(* IEC 61131-3 sources: AXOpen/src/components.kuka.robotics/ctrl/src/AxoKukaRobotics_Datatypes_v_5_x_x, 9 files *)

(* ---- AxoKukaRobotics_Component_Status.st ---- *)
NAMESPACE AXOpen.Components.Kuka.Robotics.v_5_x_x
    {S7.extern=ReadWrite}
    {#ix-attr:[Container(Layout.Stack)]}
    CLASS PUBLIC AxoKukaRobotics_Component_Status EXTENDS AXOpen.Components.Robotics.AxoRobot_Status
        VAR PUBLIC
        END_VAR
    END_CLASS
END_NAMESPACE

(* ---- AxoKukaRobotics_Component_Status_v_5_x_x.st ---- *)
NAMESPACE AXOpen.Components.Kuka.Robotics
    {S7.extern=ReadWrite}
    {#ix-attr:[Container(Layout.Stack)]}
    CLASS PUBLIC AxoKukaRobotics_Component_Status_v_5_x_x  EXTENDS AXOpen.Components.Robotics.AxoRobot_Status
        VAR PUBLIC
        END_VAR
    END_CLASS
END_NAMESPACE

(* ---- AxoKukaRobotics_Config.st ---- *)
NAMESPACE AXOpen.Components.Kuka.Robotics.v_5_x_x
    // <AxoKukaRoboticsConfigDeclaration>
    {#ix-attr:[Container(Layout.Stack)]}
    {S7.extern=ReadWrite}
    CLASS PUBLIC AxoKukaRobotics_Config
        VAR PUBLIC
            {#ix-set:AttributeName = "<#Info time#>"}
            InfoTime : LTIME := LT#2S;
            {#ix-set:AttributeName = "<#Error time#>"}
            ErrorTime : LTIME := LT#5S;
            {#ix-set:AttributeName = "<#Task timeout#>"}
            TaskTimeout : LTIME := LT#50S;
            {#ix-set:AttributeName = "<#Hardware IDs#>"}
            HWIDs : AxoKukaRobotics_HWIDs;
        END_VAR
    END_CLASS
    // </AxoKukaRoboticsConfigDeclaration>
END_NAMESPACE

(* ---- AxoKukaRobotics_Config_v_5_x_x.st ---- *)
NAMESPACE AXOpen.Components.Kuka.Robotics
    {#ix-attr:[Container(Layout.Stack)]}
    {S7.extern=ReadWrite}
    CLASS PUBLIC AxoKukaRobotics_Config_v_5_x_x
        VAR PUBLIC
            {#ix-set:AttributeName = "<#Info time#>"}
            InfoTime : LTIME := LT#2S;
            {#ix-set:AttributeName = "<#Error time#>"}
            ErrorTime : LTIME := LT#5S;
            {#ix-set:AttributeName = "<#Task timeout#>"}
            TaskTimeout : LTIME := LT#50S;
        END_VAR
    END_CLASS
END_NAMESPACE

(* ---- AxoKukaRobotics_Control.st ---- *)
NAMESPACE AXOpen.Components.Kuka.Robotics.v_5_x_x
    {S7.extern=ReadWrite}
    {#ix-attr:[Container(Layout.Wrap)]}
    CLASS AxoKukaRobotics_Control
        VAR PUBLIC
            {#ix-attr:[Container(Layout.Stack)]}
            {#ix-attr:[Group(GroupLayout.GroupBox)]}
            {#ix-set:AttributeName = "<#Program Start [EXT_START]#>"}
            ExternalStart : BOOL;
            {#ix-set:AttributeName = "<#Move Enable [MOVE_ENABLE]#>"}
            MoveEnable : BOOL;
            {#ix-set:AttributeName = "<#Error Confirmation [CONF_MESS]#>"}
            ErrorConfirmation : BOOL;
            {#ix-set:AttributeName = "<#Drives Off [DRIVES_OFF]#>"}
            DrivesOff : BOOL;
            {#ix-set:AttributeName = "<#Drives On [DRIVES_ON]#>"}
            DrivesOn : BOOL;
            {#ix-set:AttributeName = "<#Activate Interface [I_O_ACT]#>"}
            ActivateInterface : BOOL;
            {#ix-set:AttributeName = "<#Start At Main [START_AT_MAIN]#>"}
            StartAtMain : BOOL;
            {#ix-set:AttributeName = "<#Master mode#>"}
            MasterMode : BYTE;

            {#ix-attr:[Container(Layout.Stack)]}
            {#ix-attr:[Group(GroupLayout.GroupBox)]}
            {#ix-set:AttributeName = "<#Tool 1 retract#>"}
            Tool_1_Retract : BOOL;
            {#ix-set:AttributeName = "<#Tool 1 extend#>"}
            Tool_1_Extend : BOOL;
            {#ix-set:AttributeName = "<#Tool 2 retract#>"}
            Tool_2_Retract : BOOL;
            {#ix-set:AttributeName = "<#Tool 2 extend#>"}
            Tool_2_Extend : BOOL;
            {#ix-set:AttributeName = "<#Tool 3 retract#>"}
            Tool_3_Retract : BOOL;
            {#ix-set:AttributeName = "<#Tool 3 extend#>"}
            Tool_3_Extend : BOOL;
            {#ix-set:AttributeName = "<#Tool 4 retract#>"}
            Tool_4_Retract : BOOL;
            {#ix-set:AttributeName = "<#Tool 4 extend#>"}
            Tool_4_Extend : BOOL;

            {#ix-attr:[Container(Layout.Stack)]}
            {#ix-attr:[Group(GroupLayout.GroupBox)]}
            {#ix-set:AttributeName = "<#Tool 1 retract#>"}
            {#ix-set:AttributeName = "<#Zones#>"}
            Zone : BYTE;
            {#ix-set:AttributeName = "<#In position#>"}
            InPosition : BYTE;
            {#ix-set:AttributeName = "<#Action number#>"}
            ActionNo : BYTE;
            {#ix-set:AttributeName = "<#Global robot speed#>"}
            GlobalSpeed : BYTE;
            {#ix-set:AttributeName = "<#Tool number#>"}
            ToolNo : BYTE;
            {#ix-set:AttributeName = "<#Workobject number#>"}
            WorkobjectNo : BYTE;
            {#ix-set:AttributeName = "<#Point number#>"}
            PointNo : BYTE;
            {#ix-set:AttributeName = "<#User specific speed 1#>"}
            UserSpecSpeed1 : REAL;
            {#ix-set:AttributeName = "<#User specific speed 2#>"}
            UserSpecSpeed2 : REAL;

            {#ix-attr:[Container(Layout.Stack)]}
            {#ix-attr:[Group(GroupLayout.GroupBox)]}
            {attribute  addProperty Name "<#Coordinates#>"}
            Coordinates : AXOpen.Components.Abstractions.Robotics.AxoRoboticsCoordinates;
        END_VAR
    END_CLASS
END_NAMESPACE

(* ---- AxoKukaRobotics_Control_v_5_x_x.st ---- *)
NAMESPACE AXOpen.Components.Kuka.Robotics
    {S7.extern=ReadWrite}
    {#ix-attr:[Container(Layout.Wrap)]}
    CLASS AxoKukaRobotics_Control_v_5_x_x
        VAR PUBLIC
            {#ix-attr:[Container(Layout.Stack)]}
            {#ix-attr:[Group(GroupLayout.GroupBox)]}
            {#ix-set:AttributeName = "<#Program Start [EXT_START]#>"}
            ExternalStart : BOOL;
            {#ix-set:AttributeName = "<#Move Enable [MOVE_ENABLE]#>"}
            MoveEnable : BOOL;
            {#ix-set:AttributeName = "<#Error Confirmation [CONF_MESS]#>"}
            ErrorConfirmation : BOOL;
            {#ix-set:AttributeName = "<#Drives Off [DRIVES_OFF]#>"}
            DrivesOff : BOOL;
            {#ix-set:AttributeName = "<#Drives On [DRIVES_ON]#>"}
            DrivesOn : BOOL;
            {#ix-set:AttributeName = "<#Activate Interface [I_O_ACT]#>"}
            ActivateInterface : BOOL;
            {#ix-set:AttributeName = "<#Start At Main [START_AT_MAIN]#>"}
            StartAtMain : BOOL;
            {#ix-set:AttributeName = "<#Master mode#>"}
            MasterMode : BYTE;

            {#ix-attr:[Container(Layout.Stack)]}
            {#ix-attr:[Group(GroupLayout.GroupBox)]}
            {#ix-set:AttributeName = "<#Tool 1 retract#>"}
            Tool_1_Retract : BOOL;
            {#ix-set:AttributeName = "<#Tool 1 extend#>"}
            Tool_1_Extend : BOOL;
            {#ix-set:AttributeName = "<#Tool 2 retract#>"}
            Tool_2_Retract : BOOL;
            {#ix-set:AttributeName = "<#Tool 2 extend#>"}
            Tool_2_Extend : BOOL;
            {#ix-set:AttributeName = "<#Tool 3 retract#>"}
            Tool_3_Retract : BOOL;
            {#ix-set:AttributeName = "<#Tool 3 extend#>"}
            Tool_3_Extend : BOOL;
            {#ix-set:AttributeName = "<#Tool 4 retract#>"}
            Tool_4_Retract : BOOL;
            {#ix-set:AttributeName = "<#Tool 4 extend#>"}
            Tool_4_Extend : BOOL;

            {#ix-attr:[Container(Layout.Stack)]}
            {#ix-attr:[Group(GroupLayout.GroupBox)]}
            {#ix-set:AttributeName = "<#Tool 1 retract#>"}
            {#ix-set:AttributeName = "<#Zones#>"}
            Zone : BYTE;
            {#ix-set:AttributeName = "<#In position#>"}
            InPosition : BYTE;
            {#ix-set:AttributeName = "<#Action number#>"}
            ActionNo : BYTE;
            {#ix-set:AttributeName = "<#Global robot speed#>"}
            GlobalSpeed : BYTE;
            {#ix-set:AttributeName = "<#Tool number#>"}
            ToolNo : BYTE;
            {#ix-set:AttributeName = "<#Workobject number#>"}
            WorkobjectNo : BYTE;
            {#ix-set:AttributeName = "<#Point number#>"}
            PointNo : BYTE;
            {#ix-set:AttributeName = "<#User specific speed 1#>"}
            UserSpecSpeed1 : REAL;
            {#ix-set:AttributeName = "<#User specific speed 2#>"}
            UserSpecSpeed2 : REAL;

            {#ix-attr:[Container(Layout.Stack)]}
            {#ix-attr:[Group(GroupLayout.GroupBox)]}
            {attribute  addProperty Name "<#Coordinates#>"}
            Coordinates : AXOpen.Components.Abstractions.Robotics.AxoRoboticsCoordinates;
        END_VAR
    END_CLASS
END_NAMESPACE

(* ---- AxoKukaRobotics_HWIDs.st ---- *)
NAMESPACE AXOpen.Components.Kuka.Robotics.v_5_x_x
    // <AxoKukaRoboticsHWIDsDeclaration>
    {S7.extern=ReadWrite}
    {#ix-attr:[Container(Layout.Stack)]}
    CLASS PUBLIC AxoKukaRobotics_HWIDs
        VAR PUBLIC
            {#ix-set:AttributeName = "<#Hardware ID of the device#>"}
            HwID_Device            :   UINT;
            {#ix-set:AttributeName = "<#Hardware ID of the 'None' submodule#>"}
            HwID_None                :   UINT;
            {#ix-set:AttributeName = "<#Hardware ID of the '512_DI_DO' submodule#>"}
            HwID_512_DI_DO                                   :   UINT;
        END_VAR
    END_CLASS
    // </AxoKukaRoboticsHWIDsDeclaration>
END_NAMESPACE

(* ---- AxoKukaRobotics_State.st ---- *)
NAMESPACE AXOpen.Components.Kuka.Robotics.v_5_x_x
    {S7.extern=ReadWrite}
    {#ix-attr:[Container(Layout.Wrap)]}
    CLASS AxoKukaRobotics_State
        VAR PUBLIC
            {#ix-attr:[Container(Layout.Stack)]}
            {#ix-attr:[Group(GroupLayout.GroupBox)]}
            {#ix-set:AttributeName = "<#ControlReady [RC_RDY1]#>"}
            RcReady : BOOL;
            {#ix-set:AttributeName = "<#AlarmStopActive [ALARM_STOP]#>"}
            AlarmStopActive : BOOL;
            {#ix-set:AttributeName = "<#UserSafetySwitchClosed [USER_SAF]#>"}
            UserSafetySwitchClosed : BOOL;
            {#ix-set:AttributeName = "<#DrivesReady [PERI_RDY]#>"}
            DrivesReady : BOOL;
            {#ix-set:AttributeName = "<#RobotCalibrated [ROB_CAL]#>"}
            RobotCalibrated : BOOL;
            {#ix-set:AttributeName = "<#InterfaceActivated [I_O_ACTCONF]#>"}
            InterfaceActivated : BOOL;
            {#ix-set:AttributeName = "<#ErrorCollection [STOPMESS]#>"}
            StopMess : BOOL;
            {#ix-set:AttributeName = "<#RobotStopped [ROB_STOPPED]#>"}
            RobotStopped : BOOL;

            {#ix-attr:[Container(Layout.Stack)]}
            {#ix-attr:[Group(GroupLayout.GroupBox)]}
            {#ix-set:AttributeName = "<#InHome [IN_HOME]#>"}
            InHome : BOOL;
            {#ix-set:AttributeName = "<#Manual [T1]#>"}
            Manual : BOOL;
            {#ix-set:AttributeName = "<#Automatic [AUT]#>"}
            Automatic : BOOL;
            {#ix-set:AttributeName = "<#ExternalAutomatic [EXT]#>"}
            ExternalAutomatic : BOOL;
            {#ix-set:AttributeName = "<#ProcesActive [PRO_ACT]#>"}
            ProActive : BOOL;
            {#ix-set:AttributeName = "<#ProgramMoveActive [PROGRAM MOVEMENT ACTIVE]#>"}
            ProgramMoveActive : BOOL;
            {#ix-set:AttributeName = "<#Event ID#>"}
            EventId : UDINT;
            {#ix-set:AttributeName = "<#PpMoved#>"}
            PpMoved : BOOL;
            {#ix-set:AttributeName = "<#StartAtMain#>"}
            StartAtMain : BOOL;
            {#ix-set:AttributeName = "<#Error#>"}
            Error : BOOL;

            {#ix-attr:[Container(Layout.Stack)]}
            {#ix-attr:[Group(GroupLayout.GroupBox)]}
            {#ix-set:AttributeName = "<#In area 1#>"}
            InArea_1 : BOOL;
            {#ix-set:AttributeName = "<#In area 2#>"}
            InArea_2 : BOOL;
            {#ix-set:AttributeName = "<#In area 3#>"}
            InArea_3 : BOOL;
            {#ix-set:AttributeName = "<#In area 4#>"}
            InArea_4 : BOOL;
            {#ix-set:AttributeName = "<#In position 1#>"}
            InPosition_1 : BOOL;
            {#ix-set:AttributeName = "<#In position 2#>"}
            InPosition_2 : BOOL;
            {#ix-set:AttributeName = "<#In position 3#>"}
            InPosition_3 : BOOL;
            {#ix-set:AttributeName = "<#In position 4#>"}
            InPosition_4 : BOOL;
            {#ix-set:AttributeName = "<#Zones#>"}
            Zone : BYTE;
            {#ix-set:AttributeName = "<#In position#>"}
            InPosition : BYTE;

            {#ix-attr:[Container(Layout.Stack)]}
            {#ix-attr:[Group(GroupLayout.GroupBox)]}
            {#ix-set:AttributeName = "<#Tool 1 retract#>"}
            Tool_1_Retract : BOOL;
            {#ix-set:AttributeName = "<#Tool 1 extend#>"}
            Tool_1_Extend : BOOL;
            {#ix-set:AttributeName = "<#Tool 2 retract#>"}
            Tool_2_Retract : BOOL;
            {#ix-set:AttributeName = "<#Tool 2 extend#>"}
            Tool_2_Extend : BOOL;
            {#ix-set:AttributeName = "<#Tool 3 retract#>"}
            Tool_3_Retract : BOOL;
            {#ix-set:AttributeName = "<#Tool 3 extend#>"}
            Tool_3_Extend : BOOL;
            {#ix-set:AttributeName = "<#Tool 4 retract#>"}
            Tool_4_Retract : BOOL;
            {#ix-set:AttributeName = "<#Tool 4 extend#>"}
            Tool_4_Extend : BOOL;

            {#ix-attr:[Container(Layout.Stack)]}
            {#ix-attr:[Group(GroupLayout.GroupBox)]}
            {#ix-set:AttributeName = "<#Action number#>"}
            ActionNo : BYTE;
            {#ix-set:AttributeName = "<#Global speed#>"}
            GlobalSpeed : BYTE;
            {#ix-set:AttributeName = "<#Tool number#>"}
            ToolNo : BYTE;
            {#ix-set:AttributeName = "<#Workobject number#>"}
            WorkobjectNo : BYTE;
            {#ix-set:AttributeName = "<#PointNumber#>"}
            PointNo : BYTE;
            {#ix-set:AttributeName = "<#User specific speed 1#>"}
            UserSpecSpeed1 : DINT;
            {#ix-set:AttributeName = "<#User specific speed 2#>"}
            UserSpecSpeed2 : DINT;

            {#ix-attr:[Container(Layout.Stack)]}
            {#ix-attr:[Group(GroupLayout.GroupBox)]}
            {attribute  addProperty Name "<#Coordinates#>"}
            Coordinates : AXOpen.Components.Abstractions.Robotics.AxoRoboticsCoordinates;
        END_VAR
    END_CLASS
END_NAMESPACE

(* ---- AxoKukaRobotics_State_v_5_x_x.st ---- *)
NAMESPACE AXOpen.Components.Kuka.Robotics
    {S7.extern=ReadWrite}
    {#ix-attr:[Container(Layout.Wrap)]}
    CLASS AxoKukaRobotics_State_v_5_x_x
        VAR PUBLIC
            {#ix-attr:[Container(Layout.Stack)]}
            {#ix-attr:[Group(GroupLayout.GroupBox)]}
            {#ix-set:AttributeName = "<#ControlReady [RC_RDY1]#>"}
            RcReady : BOOL;
            {#ix-set:AttributeName = "<#AlarmStopActive [ALARM_STOP]#>"}
            AlarmStopActive : BOOL;
            {#ix-set:AttributeName = "<#UserSafetySwitchClosed [USER_SAF]#>"}
            UserSafetySwitchClosed : BOOL;
            {#ix-set:AttributeName = "<#DrivesReady [PERI_RDY]#>"}
            DrivesReady : BOOL;
            {#ix-set:AttributeName = "<#RobotCalibrated [ROB_CAL]#>"}
            RobotCalibrated : BOOL;
            {#ix-set:AttributeName = "<#InterfaceActivated [I_O_ACTCONF]#>"}
            InterfaceActivated : BOOL;
            {#ix-set:AttributeName = "<#ErrorCollection [STOPMESS]#>"}
            StopMess : BOOL;
            {#ix-set:AttributeName = "<#RobotStopped [ROB_STOPPED]#>"}
            RobotStopped : BOOL;

            {#ix-attr:[Container(Layout.Stack)]}
            {#ix-attr:[Group(GroupLayout.GroupBox)]}
            {#ix-set:AttributeName = "<#InHome [IN_HOME]#>"}
            InHome : BOOL;
            {#ix-set:AttributeName = "<#Manual [T1]#>"}
            Manual : BOOL;
            {#ix-set:AttributeName = "<#Automatic [AUT]#>"}
            Automatic : BOOL;
            {#ix-set:AttributeName = "<#ExternalAutomatic [EXT]#>"}
            ExternalAutomatic : BOOL;
            {#ix-set:AttributeName = "<#ProcesActive [PRO_ACT]#>"}
            ProActive : BOOL;
            {#ix-set:AttributeName = "<#ProgramMoveActive [PROGRAM MOVEMENT ACTIVE]#>"}
            ProgramMoveActive : BOOL;
            {#ix-set:AttributeName = "<#Event ID#>"}
            EventId : UDINT;
            {#ix-set:AttributeName = "<#PpMoved#>"}
            PpMoved : BOOL;
            {#ix-set:AttributeName = "<#StartAtMain#>"}
            StartAtMain : BOOL;
            {#ix-set:AttributeName = "<#Error#>"}
            Error : BOOL;

            {#ix-attr:[Container(Layout.Stack)]}
            {#ix-attr:[Group(GroupLayout.GroupBox)]}
            {#ix-set:AttributeName = "<#In area 1#>"}
            InArea_1 : BOOL;
            {#ix-set:AttributeName = "<#In area 2#>"}
            InArea_2 : BOOL;
            {#ix-set:AttributeName = "<#In area 3#>"}
            InArea_3 : BOOL;
            {#ix-set:AttributeName = "<#In area 4#>"}
            InArea_4 : BOOL;
            {#ix-set:AttributeName = "<#In position 1#>"}
            InPosition_1 : BOOL;
            {#ix-set:AttributeName = "<#In position 2#>"}
            InPosition_2 : BOOL;
            {#ix-set:AttributeName = "<#In position 3#>"}
            InPosition_3 : BOOL;
            {#ix-set:AttributeName = "<#In position 4#>"}
            InPosition_4 : BOOL;
            {#ix-set:AttributeName = "<#Zones#>"}
            Zone : BYTE;
            {#ix-set:AttributeName = "<#In position#>"}
            InPosition : BYTE;

            {#ix-attr:[Container(Layout.Stack)]}
            {#ix-attr:[Group(GroupLayout.GroupBox)]}
            {#ix-set:AttributeName = "<#Tool 1 retract#>"}
            Tool_1_Retract : BOOL;
            {#ix-set:AttributeName = "<#Tool 1 extend#>"}
            Tool_1_Extend : BOOL;
            {#ix-set:AttributeName = "<#Tool 2 retract#>"}
            Tool_2_Retract : BOOL;
            {#ix-set:AttributeName = "<#Tool 2 extend#>"}
            Tool_2_Extend : BOOL;
            {#ix-set:AttributeName = "<#Tool 3 retract#>"}
            Tool_3_Retract : BOOL;
            {#ix-set:AttributeName = "<#Tool 3 extend#>"}
            Tool_3_Extend : BOOL;
            {#ix-set:AttributeName = "<#Tool 4 retract#>"}
            Tool_4_Retract : BOOL;
            {#ix-set:AttributeName = "<#Tool 4 extend#>"}
            Tool_4_Extend : BOOL;

            {#ix-attr:[Container(Layout.Stack)]}
            {#ix-attr:[Group(GroupLayout.GroupBox)]}
            {#ix-set:AttributeName = "<#Action number#>"}
            ActionNo : BYTE;
            {#ix-set:AttributeName = "<#Global speed#>"}
            GlobalSpeed : BYTE;
            {#ix-set:AttributeName = "<#Tool number#>"}
            ToolNo : BYTE;
            {#ix-set:AttributeName = "<#Workobject number#>"}
            WorkobjectNo : BYTE;
            {#ix-set:AttributeName = "<#PointNumber#>"}
            PointNo : BYTE;
            {#ix-set:AttributeName = "<#User specific speed 1#>"}
            UserSpecSpeed1 : DINT;
            {#ix-set:AttributeName = "<#User specific speed 2#>"}
            UserSpecSpeed2 : DINT;

            {#ix-attr:[Container(Layout.Stack)]}
            {#ix-attr:[Group(GroupLayout.GroupBox)]}
            {attribute  addProperty Name "<#Coordinates#>"}
            Coordinates : AXOpen.Components.Abstractions.Robotics.AxoRoboticsCoordinates;
        END_VAR
    END_CLASS
END_NAMESPACE
